// TIA Portal V16 export
// export: Created 2022-02-09T12:05:18.4547131Z, ExportSetting WithDefaults, DisplayName Totally Integrated Automation Portal, DisplayVersion V16 Update 5, DisplayName TIA Portal Version Control Interface, DisplayVersion V16 Update 2, DisplayName TIA Portal Openness, DisplayVersion V16 Update 5, DisplayName STEP 7 Professional, DisplayVersion V16 Update 5, DisplayName STEP 7 Safety, DisplayVersion V16, DisplayName WinCC Professional, DisplayVersion V16 Update 5, DisplayName SIMATIC Visualization Architect, DisplayVersion V16
DATA_BLOCK "HmiData"   // DB3
{ S7_Optimized_Access := 'FALSE' }
VERSION : 0.1
// stored: AutoNumber false, DBAccessibleFromOPCUA true, IsOnlyStoredInLoadMemory false, IsWriteProtectedInAS false
   VAR
      getPlcMode : Int := 8;
      retValueTime : Int := 1;
      HMI_DateTime : DTL := DTL#1970-01-01-00:00:00;
      HMI_ImageNumber : Array[0..4] of Int;
      HMI_Project : Int := 0;
      PLC_Coordination : Word := 16#0000;
      PLC_DateTime : DTL := DTL#2020-06-20-20:58:39.107223992;
      PLC_Comands : Array[0..3] of Word;
      PLC_Register : Array[0..4] of Word;
   END_VAR
BEGIN
   HMI_ImageNumber[0] := 1;
   HMI_ImageNumber[1] := 102;
   HMI_ImageNumber[2..4] := 0;
   PLC_Comands[0..3] := 16#0000;
   PLC_Register[0..4] := 16#0000;
END_DATA_BLOCK
